FUNCTION_BLOCK ABSTRACT AxesBase EXTENDS TExecution IMPLEMENTS IDevice
VAR_INPUT
END_VAR
VAR_OUTPUT
END_VAR
VAR
	{attribute 'OPC.UA.DA' := '0'}
	_name : STRING;
	{attribute 'OPC.UA.DA' := '0'}
	_deviceID : STRING;					
	{attribute 'OPC.UA.DA' := '0'}
	_family : DeviceFamily;				
	{attribute 'OPC.UA.DA' := '0'}
	_logger : Logger;
	{attribute 'OPC.UA.DA' := '0'}
	_message : StringBuilder;	
	{attribute 'OPC.UA.DA' := '0'}
	_axisConfig : DeviceConfiguration;
	
	{attribute 'OPC.UA.DA' := '0'}
	_lifeTimeCount : UINT;
	{attribute 'OPC.UA.DA' := '0'}
	_notifyIsAlive : BOOL;
	{attribute 'OPC.UA.DA' := '0'}
	_pulseIsAliveGenerator : TON;
	
	StateMsg : STRING(255);
	IsAliveMsg : STRING(255);
END_VAR


// Check if it's still alive	
IF _notifyIsAlive THEN
	IsAliveMsg := TO_STRING(_lifeTimeCount);
	_notifyIsAlive := FALSE;
END_IF

IF HardwareGlobalVariables.ChamberState <> State THEN
	HardwareGlobalVariables.ChamberState := State;
	StateMsg := ANY_TO_STRING(State);		
END_IF

MessageScheduler();

PROPERTY DeviceID : STRING
GET
DeviceID := _deviceID;
END_GET
SET
_deviceID := DeviceID;
END_SET
END_PROPERTY

PROPERTY Family : DeviceFamily
GET
Family := _family;
END_GET
SET
_family := Family;
END_SET
END_PROPERTY

METHOD PROTECTED IsAlive
VAR_INPUT
END_VAR
_notifyIsAlive := TRUE;

IF _lifeTimeCount < 5 THEN
	_lifeTimeCount := _lifeTimeCount + 1;
ELSE
	_lifeTimeCount := 1;
END_IF
END_METHOD

METHOD MessageScheduler
VAR_INPUT
END_VAR
IF _pulseIsAliveGenerator.Q THEN
	_pulseIsAliveGenerator(IN := FALSE, PT := T#10MS);
		
	IsAlive();	
ELSE
	_pulseIsAliveGenerator(IN := TRUE, PT := T#1000MS);		
END_IF
END_METHOD

METHOD PROTECTED ABSTRACT MoveAbsPosition
VAR_INPUT
	Execute : BOOL;
	Position : LREAL; //EPosition;
END_VAR
END_METHOD

PROPERTY Name : STRING
GET
Name := _name;
END_GET
SET
_name := Name;
END_SET
END_PROPERTY

END_FUNCTION_BLOCK

(* stored: Version 1.1.0.1, ProductVersion 3.1.4024.12
   POU AxesBase: Id {cd5d79a4-3b04-40d7-9f56-0553f86c9b31}, SpecialFunc None
   Property DeviceID: Id {85420e8a-e4f2-47ed-a99f-b76df4867d0a}
   Get Get: Id {93855ba7-d9a0-4f5b-9054-262671711d13}
   Set Set: Id {fd86510f-f029-4453-b28b-4048865c0df2}
   Property Family: Id {55d3da33-1153-4204-84c9-7aabf7f213cb}
   Get Get: Id {53ab9884-0c85-4a3a-9a98-262f5875db83}
   Set Set: Id {7a5e9001-c6cb-4221-97e4-0ce1912270d2}
   Method IsAlive: Id {7bc9fe43-0c12-4833-a487-6e69c7dd22a3}
   Method MessageScheduler: Id {83a33768-5f62-48f2-8f97-5dc5cc3acd3f}
   Method MoveAbsPosition: Id {02a213db-72ac-4d1b-9355-861cfcdc8ce6}
   Property Name: Id {7293b69b-a59e-49ee-baf9-d41b48119af4}
   Get Get: Id {bf4b82c8-8b09-49c4-aeee-57aef09e4af7}
   Set Set: Id {6d34e5a7-6013-45ec-acd8-bbadb3535111} *)
